INTERFACE I_RpcResponse

METHOD PUBLIC Build : I_ResponseBuilder
VAR_INPUT
END_VAR
END_METHOD

METHOD PUBLIC Reject
VAR_INPUT
	Message : T_MAXSTRING;
END_VAR
END_METHOD

END_INTERFACE

(* stored: Version 1.1.0.1, ProductVersion 3.1.4024.12
   Itf I_RpcResponse: Id {3904ec60-cfb1-4857-aef6-8006191526d2}
   Method Build: Id {c09e5d3c-2fa8-4ae7-bb49-9faca20f18a1}
   Method Reject: Id {e89b7f10-45cf-41d6-88a6-c6bd74b7b997} *)
